(* Logix 5000 project; controller ARS14002_PLC vendor 1 type 14 code 218 rev 30.11; software revision 30.01; part 7 of 13 *)
(* tags used below, declared in another part *)
   AN_1000A : CM_AI_SCL;
   AN_1000A_SP : REAL;
   AN_1000A_SPL : REAL;
   AN_1000B : CM_AI_SCL;
   AN_1000B_SP : REAL;
   AN_1000B_SPL : REAL;
   ARGON_FROM_TK1100A : BOOL;
   ARGON_FROM_TK700 : BOOL;
   ARS_DERIME_AUTO : BOOL;
   ARS_RETURN : BOOL;
   ARS_RETURN_AUTO : BOOL;
   ARS_SOURCE_SWITCH_AUTO : BOOL;   // Switch between TK-700 and TK-1100A
   ARS_STANDBY : BOOL;
   AT2_PLANT_BACKFILL : BOOL;
   AT2_PLANT_RETURN_AUTO : BOOL;
   AT3_PLANT_BACKFILL : BOOL;
   AT3_PLANT_RETURN_AUTO : BOOL;
   Auto_CP_Select_HMI : BOOL;
   Auto_CP_Select_Inactive_ONS : BOOL;
   CP_Hi_Press_Shutoff : BOOL;
   CP_PumpUp : BOOL;
   CP_PumpUp_DN_ONS_OB : BOOL;
   CP_Run_Atomize : BOOL;
   CP_Run_ONS_OB : BOOL;
   CP_Run_ONS_SB : BOOL;
   CP_Run_Standby : BOOL;
   CP_Select_Auto : BOOL;
   CP_Select_Auto_ONS : BOOL;
   CP_Stop : BOOL;
   CP_Stop_ONS_OB : BOOL;
   CP_Stop_ONS_SB : BOOL;
   DERIME_HOLD : BOOL;
   ESTOP_TRIP : BOOL;
   ew_TEST_P800A_LOCKOUT : BOOL;
   FCV_753_SP_Idle : REAL;
   FCV_753_SP_Standby : REAL;
   FCV_754_SP_Idle : REAL;
   FCV_754_SP_Standby : REAL;
   FIRST_SCAN_BIT : BOOL;
   FT_904 : CM_AI_SCL;
   FVR_800C_Auto : BOOL;
   FVR_800C_Auto_ONS : BOOL;
   FVR_800C_AutoReq : BOOL;
   FVR_800C_ClearFault_TMR : TIMER;
   FVR_800C_DISABLE_ONS : BOOL;
   FVR_800C_EN : BOOL;
   FVR_800C_ManReq : BOOL;
   FVR_800C_ManStartReq : BOOL;
   FVR_800C_PRIMARY : BOOL;
   FVR_800C_RUNNING : BOOL;
   FVR_800C_ST : BOOL;
   FVR_800D_Auto : BOOL;
   FVR_800D_Auto_ONS : BOOL;
   FVR_800D_AutoReq : BOOL;
   FVR_800D_ClearFault_TMR : TIMER;
   FVR_800D_DISABLE_ONS : BOOL;
   FVR_800D_EN : BOOL;
   FVR_800D_ManReq : BOOL;
   FVR_800D_ManStartReq : BOOL;
   FVR_800D_PRIMARY : BOOL;
   FVR_800D_RUNNING : BOOL;
   FVR_800D_ST : BOOL;
   MODE_ATOMIZE : BOOL;
   MODE_IDLE : BOOL;
   MODE_STANDBY_IDLE : BOOL;
   MODE_STANDBY_PUMPUP : BOOL;
   P_800A_Cavit : BOOL;
   P_800A_Cooldown_Complete : BOOL;
   P_800A_Hi_Press_Shutoff : BOOL;
   P_800A_Init_OK : BOOL;
   P_800A_Pre_Vent_Done : BOOL;
   P_800A_Pre_Vent_Pending : BOOL;
   P_800A_Prestart : BOOL;
   P_800A_Ready : BOOL;
   P_800A_RUN_OCCURRED : BOOL;
   P_800A_Select_Auto_Online : BOOL;
   P_800A_Start_DLA_TMR : TIMER;
   P_800A_Start_Temp_SP : DINT;
   P_800A_Start_TMR : TIMER;
   P_800A_STOP_ONS : BOOL;
   P_800A_Stop_Vent_Delay : BOOL;
   P_800B_Cavit : BOOL;
   P_800B_Cooldown_Complete : BOOL;
   P_800B_Hi_Press_Shutoff : BOOL;
   P_800B_Init_OK : BOOL;
   P_800B_Pre_Vent_Done : BOOL;
   P_800B_Pre_Vent_Pending : BOOL;
   P_800B_Prestart : BOOL;
   P_800B_Ready : BOOL;
   P_800B_RUN_OCCURRED : BOOL;
   P_800B_Select_Auto_Online : BOOL;
   P_800B_Start_DLA_TMR : TIMER;
   P_800B_Start_Temp_SP : DINT;
   P_800B_Start_TMR : TIMER;
   P_800B_STOP_ONS : BOOL;
   P_800B_Stop_Vent_Delay : BOOL;
   P_800C : CM_DO_FVR;
   P_800C_Cavit : BOOL;
   P_800C_Cooldown_Complete : BOOL;
   P_800C_Fault : BOOL;
   P_800C_Hi_Press_Shutoff : BOOL;
   P_800C_Init_OK : BOOL;
   P_800C_Pre_Vent_Done : BOOL;
   P_800C_Pre_Vent_Pending : BOOL;
   P_800C_Prestart : BOOL;
   P_800C_Ready : BOOL;
   P_800C_RUN_OCCURRED : BOOL;
   P_800C_Select_Auto_Online : BOOL;
   P_800C_Start_DLA_TMR : TIMER;
   P_800C_Start_Temp_SP : DINT;
   P_800C_Start_TMR : TIMER;
   P_800C_STOP_ONS : BOOL;
   P_800C_Stop_Vent_Delay : BOOL;
   P_800D : CM_DO_FVR;
   P_800D_Cavit : BOOL;
   P_800D_Cooldown_Complete : BOOL;
   P_800D_Fault : BOOL;
   P_800D_Hi_Press_Shutoff : BOOL;
   P_800D_Init_OK : BOOL;
   P_800D_Pre_Vent_Done : BOOL;
   P_800D_Pre_Vent_Pending : BOOL;
   P_800D_Prestart : BOOL;
   P_800D_Ready : BOOL;
   P_800D_RUN_OCCURRED : BOOL;
   P_800D_Select_Auto_Online : BOOL;
   P_800D_Start_DLA_TMR : TIMER;
   P_800D_Start_TMR : TIMER;
   P_800D_STOP_ONS : BOOL;
   P_800D_Stop_Vent_Delay : BOOL;
   PDT_601 : CM_AI_SCL_ALT;
   PDT_701_ALT_GAL : REAL;
   PDT_751 : CM_AI_SCL_ALT;
   PIDE_753 : PID_ENHANCED;
   PIDE_754 : PID_ENHANCED;
   PIDE_755 : PID_ENHANCED;
   PIDE_800 : PID_ENHANCED;
   PILOT_PLANT_BACKFILL : BOOL;
   PILOT_PLANT_BACKFILL_COOLDOWN_DLA_SEC : REAL;
   PILOT_PLANT_BACKFILL_COOLDOWN_DLA_TMR : TIMER;   // delays the cooldown for a backfill
   PILOT_PLANT_RETURN_AUTO : BOOL;
   PT_751 : CM_AI_SCL;
   REQUEST_ARGON_FROM_TK1100A : BOOL;
   REQUEST_ARGON_FROM_TK700 : BOOL;
   SV_753F : CM_DO_GENERIC;
   SV_754F : CM_DO_GENERIC;
   SV_755F : CM_DO_GENERIC;
   TE_803_XV_721A_BURP_SP : REAL;
   TE_803A : CM_AI_SCL;
   TE_803B : CM_AI_SCL;
   TE_803C : CM_AI_SCL;
   TE_803D : CM_AI_SCL;
   TE_902 : CM_AI_SCL;
   TE_904 : CM_AI_SCL;
   TE_T_Fail_Temp : DINT;
   TEST_COOLDOWN_ALT : BOOL;
   TK_1100A_Low : BOOL;
   TK_700_AUTOFILL : BOOL;   // 1= TK-1100A WILL FILL TK-700
   TK_700_AUTOFILL_PDT_601_ALT_SPH : REAL;
   TK_700_AUTOFILL_SPH : REAL;
   TK_700_AUTOFILL_SPL : REAL;
   TK_700_AUTOSOURCE_SPH : REAL;   // Level where source will switch back to TK-700
   TK_700_AUTOSOURCE_SPL : REAL;   // Level where source will switch away from TK-700
   TK_700_FILLREQ : BOOL;
   TK_700_Full : BOOL;
   TK_700_Low : BOOL;
   VFD_800A_Auto : BOOL;
   VFD_800A_Auto_ONS : BOOL;
   VFD_800A_AutoReq : BOOL;
   VFD_800A_ClearFault_TMR : TIMER;
   VFD_800A_DISABLE_ONS : BOOL;
   VFD_800A_EN : BOOL;
   VFD_800A_ManReq : BOOL;
   VFD_800A_ManStartReq : BOOL;
   VFD_800A_ST : BOOL;
   VFD_800B_Auto : BOOL;
   VFD_800B_Auto_ONS : BOOL;
   VFD_800b_AutoReq : BOOL;
   VFD_800B_ClearFault_TMR : TIMER;
   VFD_800B_DISABLE_ONS : BOOL;
   VFD_800B_EN : BOOL;
   VFD_800B_ManReq : BOOL;
   VFD_800B_ManStartReq : BOOL;
   VFD_800B_ST : BOOL;
   XV_1123 : CM_DO_VLV;
   XV_703 : CM_DO_VLV;
   XV_721_BURP_AUTO : BOOL;
   XV_721A : CM_DO_VLV;
   XV_721B : CM_DO_VLV;
   XV_801A : CM_DO_VLV;
   XV_801B : CM_DO_VLV;
   XV_801C : CM_DO_VLV;
   XV_801D : CM_DO_VLV;
(* MainProgram, continued *)

ROUTINE _304_Subcooler   (* ladder *)
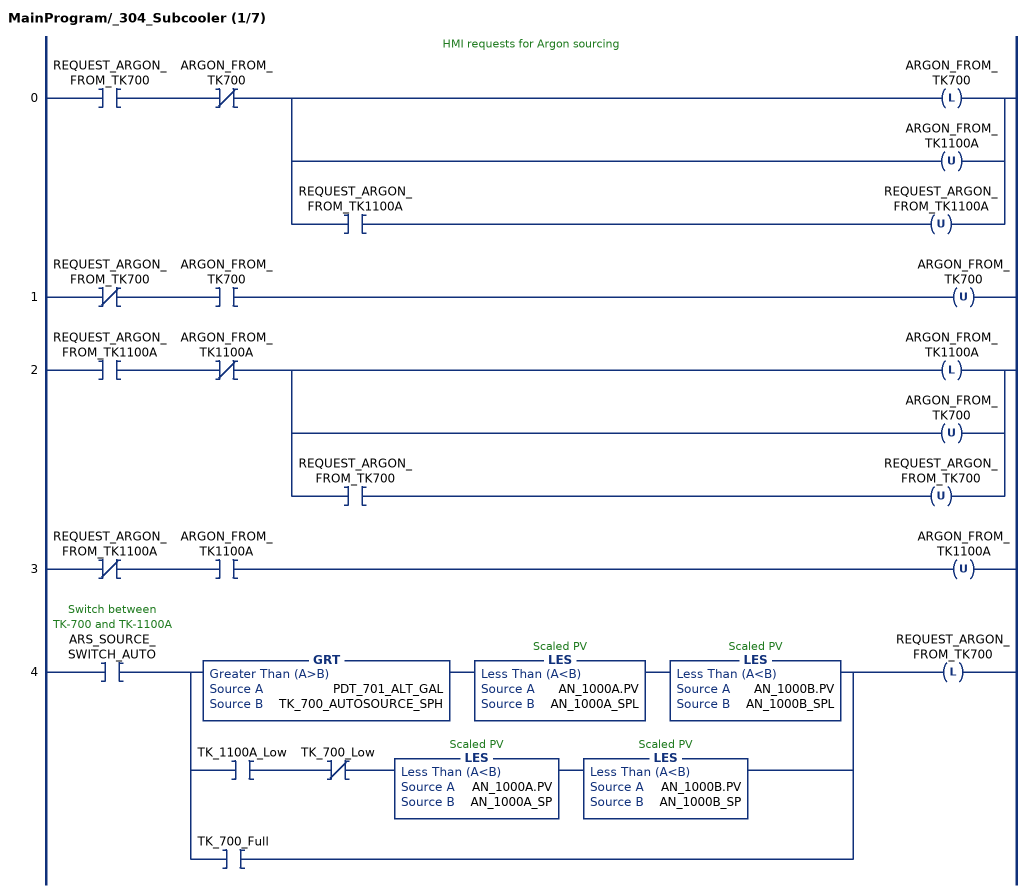
   // HMI requests for Argon sourcing
   0: XIC(REQUEST_ARGON_FROM_TK700)XIO(ARGON_FROM_TK700)[OTL(ARGON_FROM_TK700) ,OTU(ARGON_FROM_TK1100A) ,XIC(REQUEST_ARGON_FROM_TK1100A) OTU(REQUEST_ARGON_FROM_TK1100A) ];
   1: XIO(REQUEST_ARGON_FROM_TK700)XIC(ARGON_FROM_TK700)OTU(ARGON_FROM_TK700);
   2: XIC(REQUEST_ARGON_FROM_TK1100A)XIO(ARGON_FROM_TK1100A)[OTL(ARGON_FROM_TK1100A) ,OTU(ARGON_FROM_TK700) ,XIC(REQUEST_ARGON_FROM_TK700) OTU(REQUEST_ARGON_FROM_TK700) ];
   3: XIO(REQUEST_ARGON_FROM_TK1100A)XIC(ARGON_FROM_TK1100A)OTU(ARGON_FROM_TK1100A);
   4: XIC(ARS_SOURCE_SWITCH_AUTO)[GRT(PDT_701_ALT_GAL,TK_700_AUTOSOURCE_SPH) LES(AN_1000A.PV,AN_1000A_SPL) LES(AN_1000B.PV,AN_1000B_SPL) ,XIC(TK_1100A_Low) XIO(TK_700_Low) LES(AN_1000A.PV,AN_1000A_SP) LES(AN_1000B.PV,AN_1000B_SP) ,XIC(TK_700_Full) ]OTL(REQUEST_ARGON_FROM_TK700);
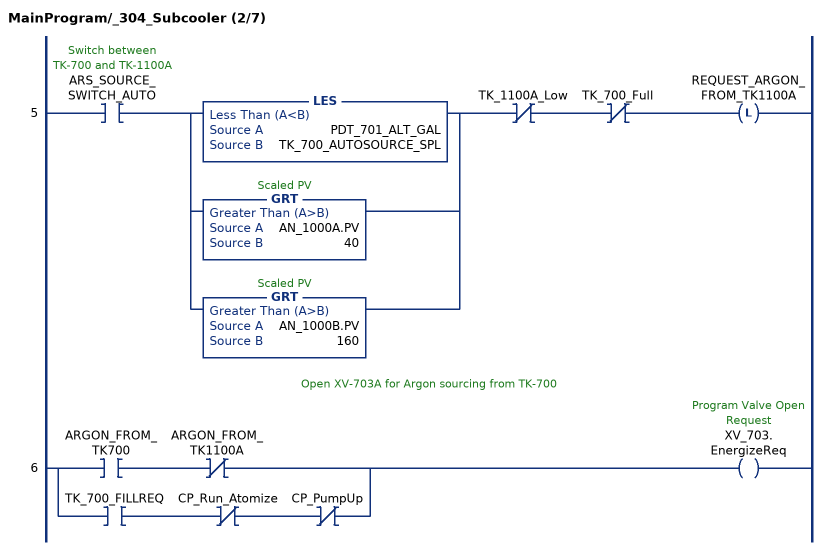
   5: XIC(ARS_SOURCE_SWITCH_AUTO)[LES(PDT_701_ALT_GAL,TK_700_AUTOSOURCE_SPL) ,GRT(AN_1000A.PV,40) ,GRT(AN_1000B.PV,160) ]XIO(TK_1100A_Low)XIO(TK_700_Full)OTL(REQUEST_ARGON_FROM_TK1100A);
   // Open XV-703A for Argon sourcing from TK-700
   6: [XIC(ARGON_FROM_TK700) XIO(ARGON_FROM_TK1100A) ,XIC(TK_700_FILLREQ) XIO(CP_Run_Atomize) XIO(CP_PumpUp) ]OTE(XV_703.EnergizeReq);
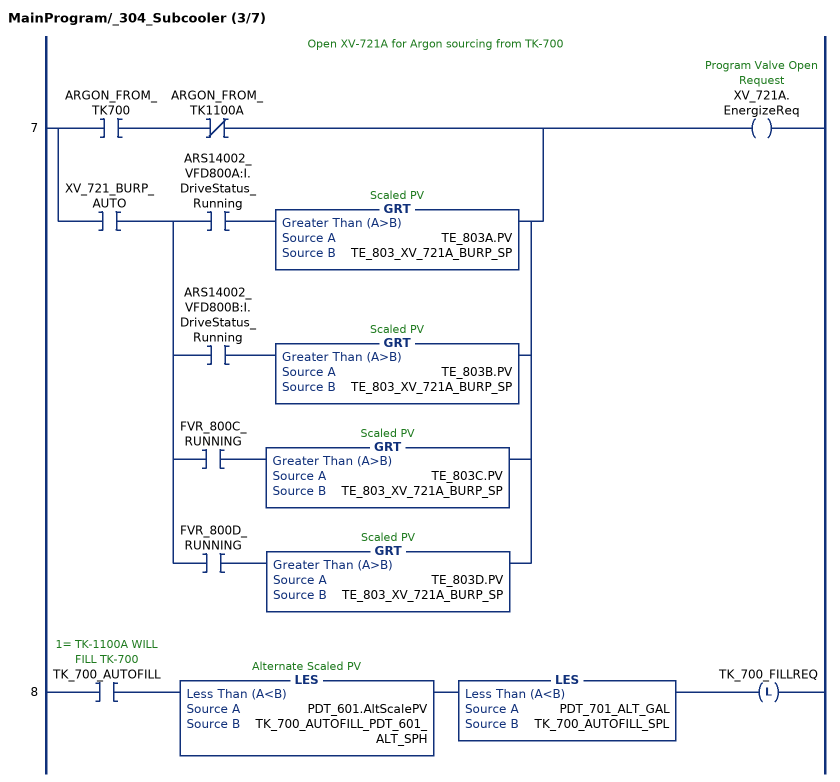
   // Open XV-721A for Argon sourcing from TK-700
   7: [XIC(ARGON_FROM_TK700) XIO(ARGON_FROM_TK1100A) ,XIC(XV_721_BURP_AUTO) [XIC(ARS14002_VFD800A:I.DriveStatus_Running) GRT(TE_803A.PV,TE_803_XV_721A_BURP_SP) ,XIC(ARS14002_VFD800B:I.DriveStatus_Running) GRT(TE_803B.PV,TE_803_XV_721A_BURP_SP) ,XIC(FVR_800C_RUNNING) GRT(TE_803C.PV,TE_803_XV_721A_BURP_SP) ,XIC(FVR_800D_RUNNING) GRT(TE_803D.PV,TE_803_XV_721A_BURP_SP) ] ]OTE(XV_721A.EnergizeReq);
   8: XIC(TK_700_AUTOFILL)LES(PDT_601.AltScalePV,TK_700_AUTOFILL_PDT_601_ALT_SPH)LES(PDT_701_ALT_GAL,TK_700_AUTOFILL_SPL)OTL(TK_700_FILLREQ);
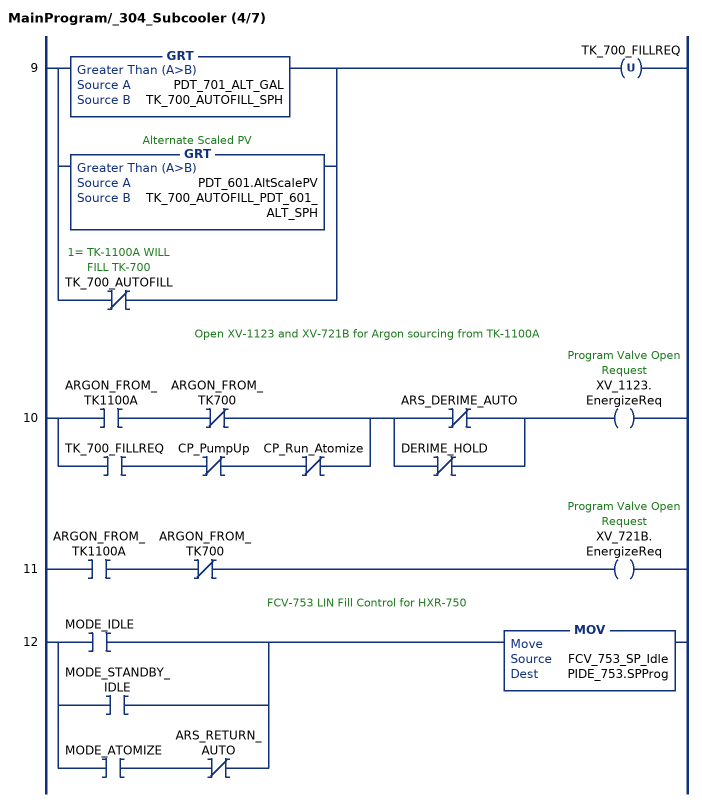
   9: [GRT(PDT_701_ALT_GAL,TK_700_AUTOFILL_SPH) ,GRT(PDT_601.AltScalePV,TK_700_AUTOFILL_PDT_601_ALT_SPH) ,XIO(TK_700_AUTOFILL) ]OTU(TK_700_FILLREQ);
   // Open XV-1123 and XV-721B for Argon sourcing from TK-1100A
   10: [XIC(ARGON_FROM_TK1100A) XIO(ARGON_FROM_TK700) ,XIC(TK_700_FILLREQ) XIO(CP_PumpUp) XIO(CP_Run_Atomize) ][XIO(ARS_DERIME_AUTO) ,XIO(DERIME_HOLD) ]OTE(XV_1123.EnergizeReq);
   11: XIC(ARGON_FROM_TK1100A)XIO(ARGON_FROM_TK700)OTE(XV_721B.EnergizeReq);
   // FCV-753 LIN Fill Control for HXR-750
   12: [XIC(MODE_IDLE) ,XIC(MODE_STANDBY_IDLE) ,XIC(MODE_ATOMIZE) XIO(ARS_RETURN_AUTO) ]MOV(FCV_753_SP_Idle,PIDE_753.SPProg);
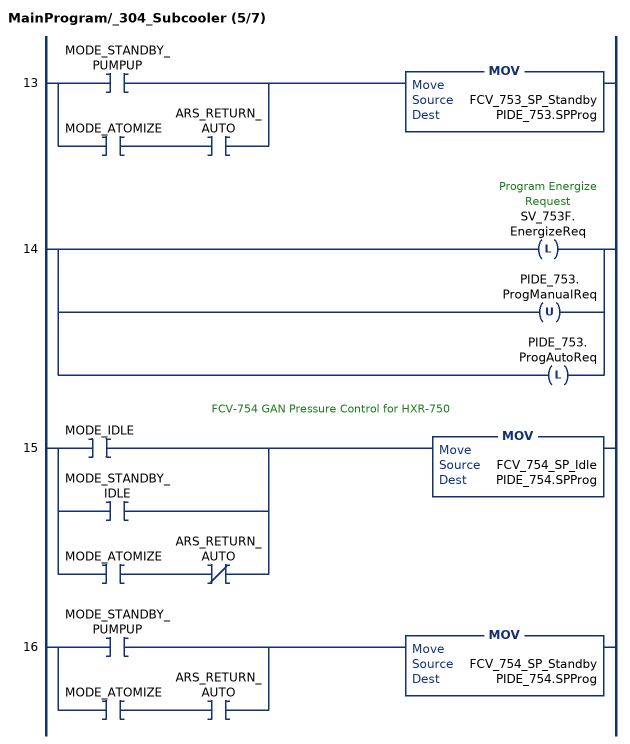
   13: [XIC(MODE_STANDBY_PUMPUP) ,XIC(MODE_ATOMIZE) XIC(ARS_RETURN_AUTO) ]MOV(FCV_753_SP_Standby,PIDE_753.SPProg);
   14: [OTL(SV_753F.EnergizeReq) ,OTU(PIDE_753.ProgManualReq) ,OTL(PIDE_753.ProgAutoReq) ];
   // FCV-754 GAN Pressure Control for HXR-750
   15: [XIC(MODE_IDLE) ,XIC(MODE_STANDBY_IDLE) ,XIC(MODE_ATOMIZE) XIO(ARS_RETURN_AUTO) ]MOV(FCV_754_SP_Idle,PIDE_754.SPProg);
   16: [XIC(MODE_STANDBY_PUMPUP) ,XIC(MODE_ATOMIZE) XIC(ARS_RETURN_AUTO) ]MOV(FCV_754_SP_Standby,PIDE_754.SPProg);
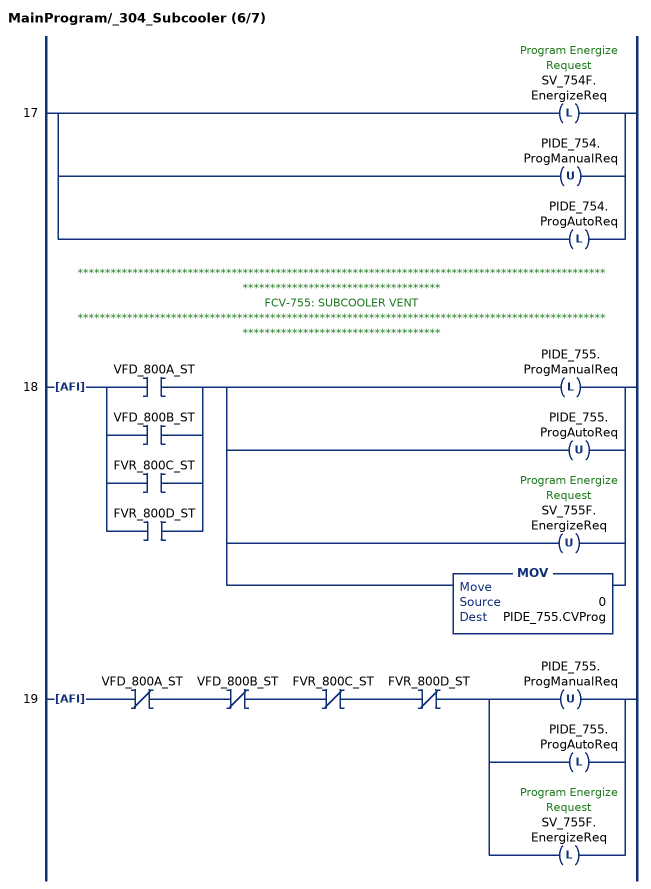
   17: [OTL(SV_754F.EnergizeReq) ,OTU(PIDE_754.ProgManualReq) ,OTL(PIDE_754.ProgAutoReq) ];
   // ************************************************************************************************************************************
   // FCV-755: SUBCOOLER VENT
   // ************************************************************************************************************************************
   18: AFI()[XIC(VFD_800A_ST) ,XIC(VFD_800B_ST) ,XIC(FVR_800C_ST) ,XIC(FVR_800D_ST) ][OTL(PIDE_755.ProgManualReq) ,OTU(PIDE_755.ProgAutoReq) ,OTU(SV_755F.EnergizeReq) ,MOV(0,PIDE_755.CVProg) ];
   19: AFI()XIO(VFD_800A_ST)XIO(VFD_800B_ST)XIO(FVR_800C_ST)XIO(FVR_800D_ST)[OTU(PIDE_755.ProgManualReq) ,OTL(PIDE_755.ProgAutoReq) ,OTL(SV_755F.EnergizeReq) ];
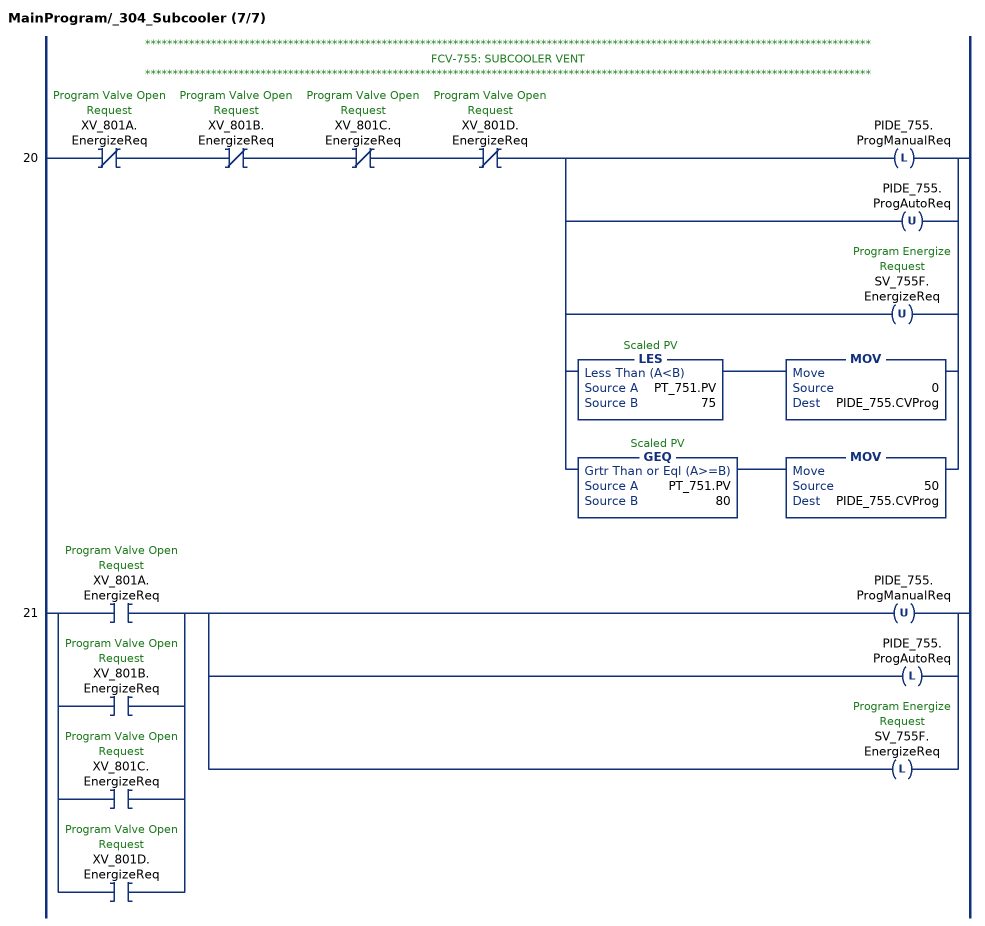
   // ************************************************************************************************************************************
   // FCV-755: SUBCOOLER VENT
   // ************************************************************************************************************************************
   20: XIO(XV_801A.EnergizeReq)XIO(XV_801B.EnergizeReq)XIO(XV_801C.EnergizeReq)XIO(XV_801D.EnergizeReq)[OTL(PIDE_755.ProgManualReq) ,OTU(PIDE_755.ProgAutoReq) ,OTU(SV_755F.EnergizeReq) ,LES(PT_751.PV,75) MOV(0,PIDE_755.CVProg) ,GEQ(PT_751.PV,80) MOV(50,PIDE_755.CVProg) ];
   21: [XIC(XV_801A.EnergizeReq) ,XIC(XV_801B.EnergizeReq) ,XIC(XV_801C.EnergizeReq) ,XIC(XV_801D.EnergizeReq) ][OTU(PIDE_755.ProgManualReq) ,OTL(PIDE_755.ProgAutoReq) ,OTL(SV_755F.EnergizeReq) ];
END_ROUTINE

ROUTINE _305_Pump_800   (* ladder *)
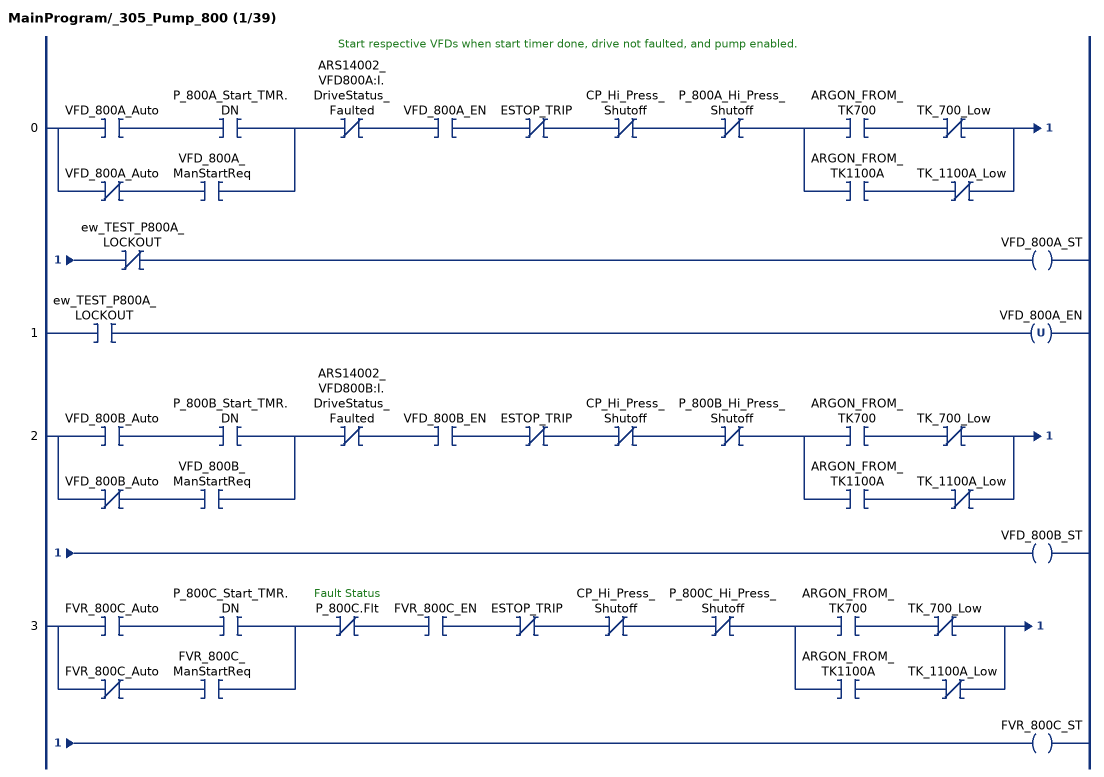
   // Start respective VFDs when start timer done, drive not faulted, and pump enabled.
   0: [XIC(VFD_800A_Auto) XIC(P_800A_Start_TMR.DN) ,XIO(VFD_800A_Auto) XIC(VFD_800A_ManStartReq) ]XIO(ARS14002_VFD800A:I.DriveStatus_Faulted)XIC(VFD_800A_EN)XIO(ESTOP_TRIP)XIO(CP_Hi_Press_Shutoff)XIO(P_800A_Hi_Press_Shutoff)[XIC(ARGON_FROM_TK700) XIO(TK_700_Low) ,XIC(ARGON_FROM_TK1100A) XIO(TK_1100A_Low) ]XIO(ew_TEST_P800A_LOCKOUT)OTE(VFD_800A_ST);
   1: XIC(ew_TEST_P800A_LOCKOUT)OTU(VFD_800A_EN);
   2: [XIC(VFD_800B_Auto) XIC(P_800B_Start_TMR.DN) ,XIO(VFD_800B_Auto) XIC(VFD_800B_ManStartReq) ]XIO(ARS14002_VFD800B:I.DriveStatus_Faulted)XIC(VFD_800B_EN)XIO(ESTOP_TRIP)XIO(CP_Hi_Press_Shutoff)XIO(P_800B_Hi_Press_Shutoff)[XIC(ARGON_FROM_TK700) XIO(TK_700_Low) ,XIC(ARGON_FROM_TK1100A) XIO(TK_1100A_Low) ]OTE(VFD_800B_ST);
   3: [XIC(FVR_800C_Auto) XIC(P_800C_Start_TMR.DN) ,XIO(FVR_800C_Auto) XIC(FVR_800C_ManStartReq) ]XIO(P_800C.Flt)XIC(FVR_800C_EN)XIO(ESTOP_TRIP)XIO(CP_Hi_Press_Shutoff)XIO(P_800C_Hi_Press_Shutoff)[XIC(ARGON_FROM_TK700) XIO(TK_700_Low) ,XIC(ARGON_FROM_TK1100A) XIO(TK_1100A_Low) ]OTE(FVR_800C_ST);
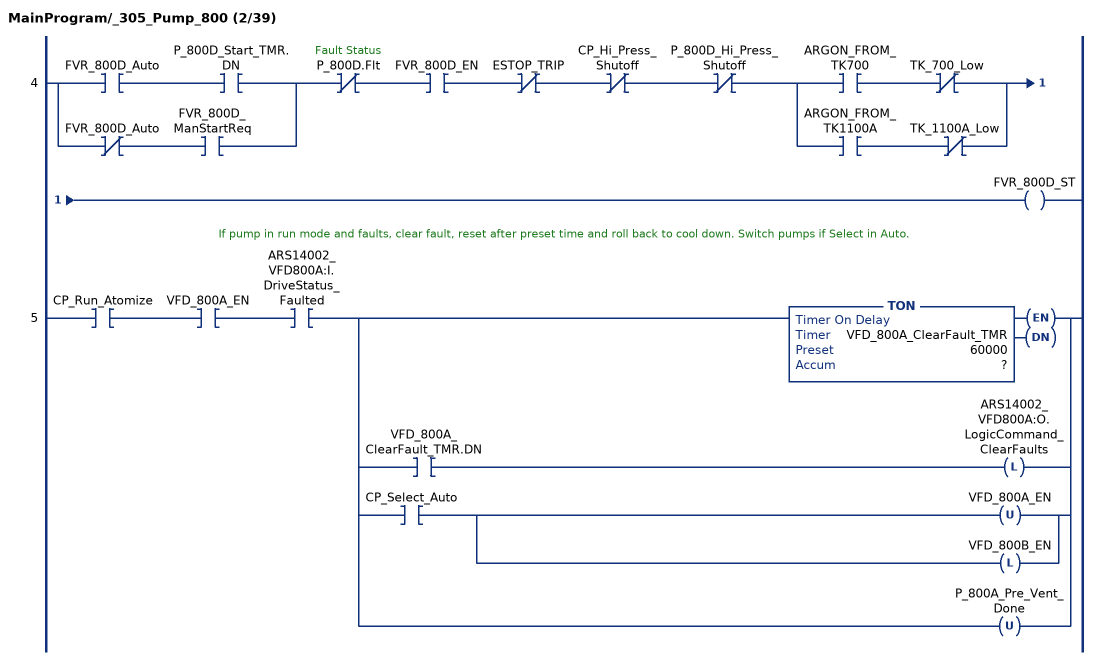
   4: [XIC(FVR_800D_Auto) XIC(P_800D_Start_TMR.DN) ,XIO(FVR_800D_Auto) XIC(FVR_800D_ManStartReq) ]XIO(P_800D.Flt)XIC(FVR_800D_EN)XIO(ESTOP_TRIP)XIO(CP_Hi_Press_Shutoff)XIO(P_800D_Hi_Press_Shutoff)[XIC(ARGON_FROM_TK700) XIO(TK_700_Low) ,XIC(ARGON_FROM_TK1100A) XIO(TK_1100A_Low) ]OTE(FVR_800D_ST);
   // If pump in run mode and faults, clear fault, reset after preset time and roll back to cool down. Switch pumps if Select in Auto.
   5: XIC(CP_Run_Atomize)XIC(VFD_800A_EN)XIC(ARS14002_VFD800A:I.DriveStatus_Faulted)[[TON(VFD_800A_ClearFault_TMR,?,?) ,XIC(VFD_800A_ClearFault_TMR.DN) OTL(ARS14002_VFD800A:O.LogicCommand_ClearFaults) ,XIC(CP_Select_Auto) [OTU(VFD_800A_EN) ,OTL(VFD_800B_EN) ] ] ,OTU(P_800A_Pre_Vent_Done) ];
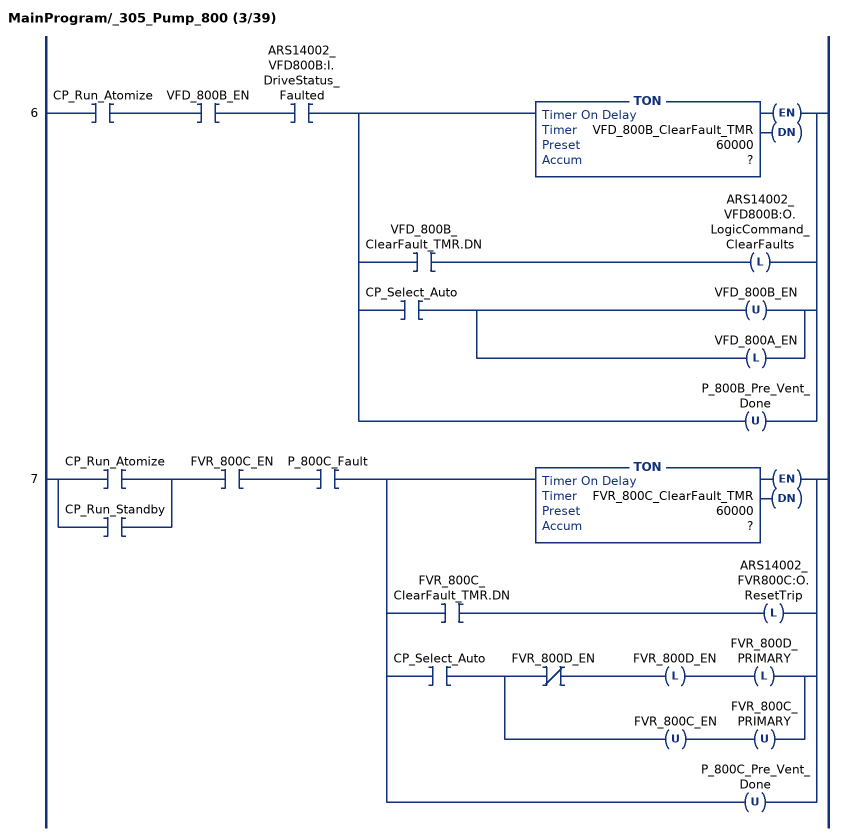
   6: XIC(CP_Run_Atomize)XIC(VFD_800B_EN)XIC(ARS14002_VFD800B:I.DriveStatus_Faulted)[[TON(VFD_800B_ClearFault_TMR,?,?) ,XIC(VFD_800B_ClearFault_TMR.DN) OTL(ARS14002_VFD800B:O.LogicCommand_ClearFaults) ,XIC(CP_Select_Auto) [OTU(VFD_800B_EN) ,OTL(VFD_800A_EN) ] ] ,OTU(P_800B_Pre_Vent_Done) ];
   7: [XIC(CP_Run_Atomize) ,XIC(CP_Run_Standby) ]XIC(FVR_800C_EN)XIC(P_800C_Fault)[[TON(FVR_800C_ClearFault_TMR,?,?) ,XIC(FVR_800C_ClearFault_TMR.DN) OTL(ARS14002_FVR800C:O.ResetTrip) ,XIC(CP_Select_Auto) [XIO(FVR_800D_EN) OTL(FVR_800D_EN) OTL(FVR_800D_PRIMARY) ,OTU(FVR_800C_EN) OTU(FVR_800C_PRIMARY) ] ] ,OTU(P_800C_Pre_Vent_Done) ];
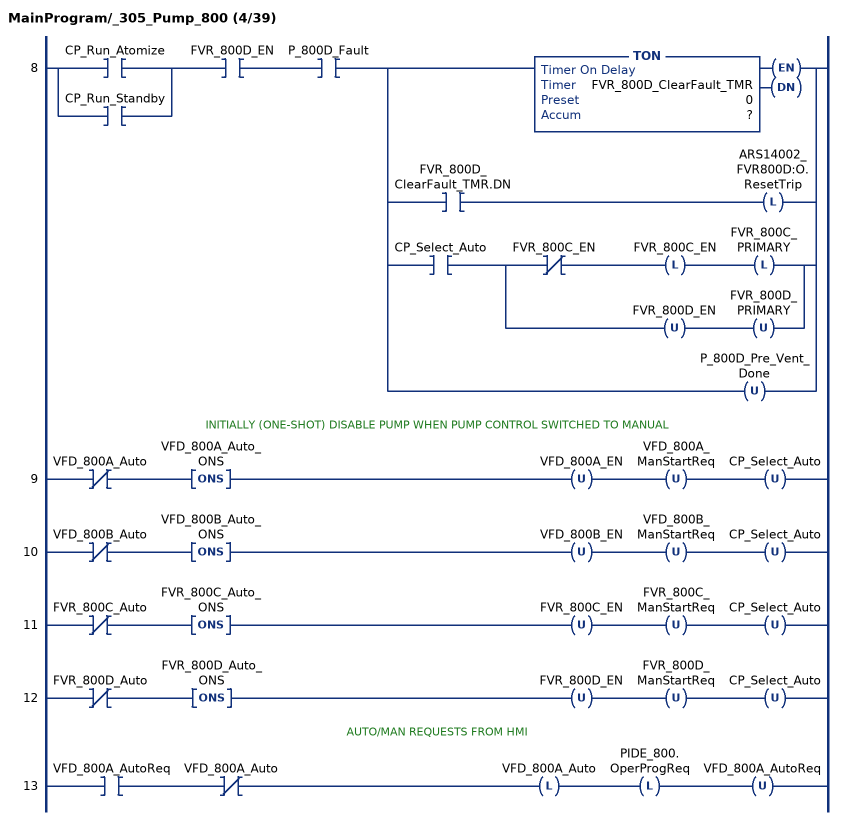
   8: [XIC(CP_Run_Atomize) ,XIC(CP_Run_Standby) ]XIC(FVR_800D_EN)XIC(P_800D_Fault)[[TON(FVR_800D_ClearFault_TMR,?,?) ,XIC(FVR_800D_ClearFault_TMR.DN) OTL(ARS14002_FVR800D:O.ResetTrip) ,XIC(CP_Select_Auto) [XIO(FVR_800C_EN) OTL(FVR_800C_EN) OTL(FVR_800C_PRIMARY) ,OTU(FVR_800D_EN) OTU(FVR_800D_PRIMARY) ] ] ,OTU(P_800D_Pre_Vent_Done) ];
   // INITIALLY (ONE-SHOT) DISABLE PUMP WHEN PUMP CONTROL SWITCHED TO MANUAL
   9: XIO(VFD_800A_Auto)ONS(VFD_800A_Auto_ONS)OTU(VFD_800A_EN)OTU(VFD_800A_ManStartReq)OTU(CP_Select_Auto);
   10: XIO(VFD_800B_Auto)ONS(VFD_800B_Auto_ONS)OTU(VFD_800B_EN)OTU(VFD_800B_ManStartReq)OTU(CP_Select_Auto);
   11: XIO(FVR_800C_Auto)ONS(FVR_800C_Auto_ONS)OTU(FVR_800C_EN)OTU(FVR_800C_ManStartReq)OTU(CP_Select_Auto);
   12: XIO(FVR_800D_Auto)ONS(FVR_800D_Auto_ONS)OTU(FVR_800D_EN)OTU(FVR_800D_ManStartReq)OTU(CP_Select_Auto);
   // AUTO/MAN REQUESTS FROM HMI
   13: XIC(VFD_800A_AutoReq)XIO(VFD_800A_Auto)OTL(VFD_800A_Auto)OTL(PIDE_800.OperProgReq)OTU(VFD_800A_AutoReq);
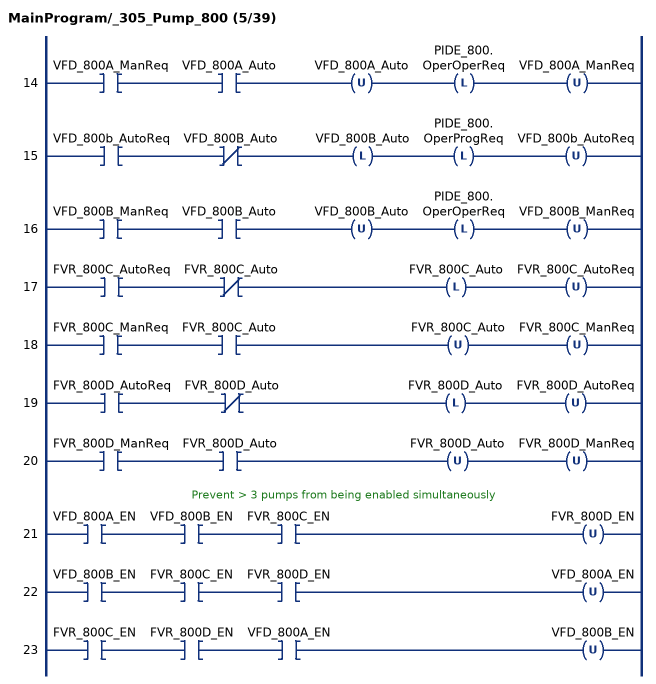
   14: XIC(VFD_800A_ManReq)XIC(VFD_800A_Auto)OTU(VFD_800A_Auto)OTL(PIDE_800.OperOperReq)OTU(VFD_800A_ManReq);
   15: XIC(VFD_800b_AutoReq)XIO(VFD_800B_Auto)OTL(VFD_800B_Auto)OTL(PIDE_800.OperProgReq)OTU(VFD_800b_AutoReq);
   16: XIC(VFD_800B_ManReq)XIC(VFD_800B_Auto)OTU(VFD_800B_Auto)OTL(PIDE_800.OperOperReq)OTU(VFD_800B_ManReq);
   17: XIC(FVR_800C_AutoReq)XIO(FVR_800C_Auto)OTL(FVR_800C_Auto)OTU(FVR_800C_AutoReq);
   18: XIC(FVR_800C_ManReq)XIC(FVR_800C_Auto)OTU(FVR_800C_Auto)OTU(FVR_800C_ManReq);
   19: XIC(FVR_800D_AutoReq)XIO(FVR_800D_Auto)OTL(FVR_800D_Auto)OTU(FVR_800D_AutoReq);
   20: XIC(FVR_800D_ManReq)XIC(FVR_800D_Auto)OTU(FVR_800D_Auto)OTU(FVR_800D_ManReq);
   // Prevent > 3 pumps from being enabled simultaneously
   21: XIC(VFD_800A_EN)XIC(VFD_800B_EN)XIC(FVR_800C_EN)OTU(FVR_800D_EN);
   22: XIC(VFD_800B_EN)XIC(FVR_800C_EN)XIC(FVR_800D_EN)OTU(VFD_800A_EN);
   23: XIC(FVR_800C_EN)XIC(FVR_800D_EN)XIC(VFD_800A_EN)OTU(VFD_800B_EN);
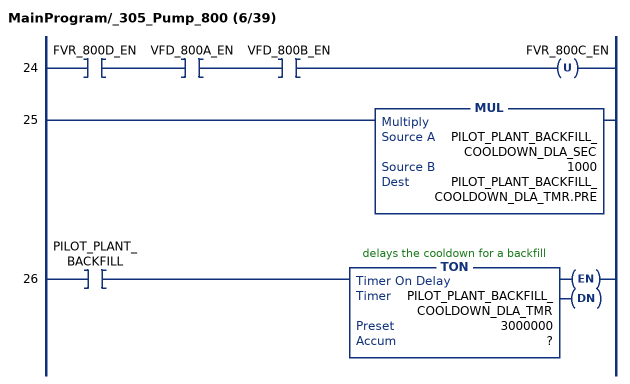
   24: XIC(FVR_800D_EN)XIC(VFD_800A_EN)XIC(VFD_800B_EN)OTU(FVR_800C_EN);
   25: MUL(PILOT_PLANT_BACKFILL_COOLDOWN_DLA_SEC,1000,PILOT_PLANT_BACKFILL_COOLDOWN_DLA_TMR.PRE);
   26: XIC(PILOT_PLANT_BACKFILL)TON(PILOT_PLANT_BACKFILL_COOLDOWN_DLA_TMR,?,?);
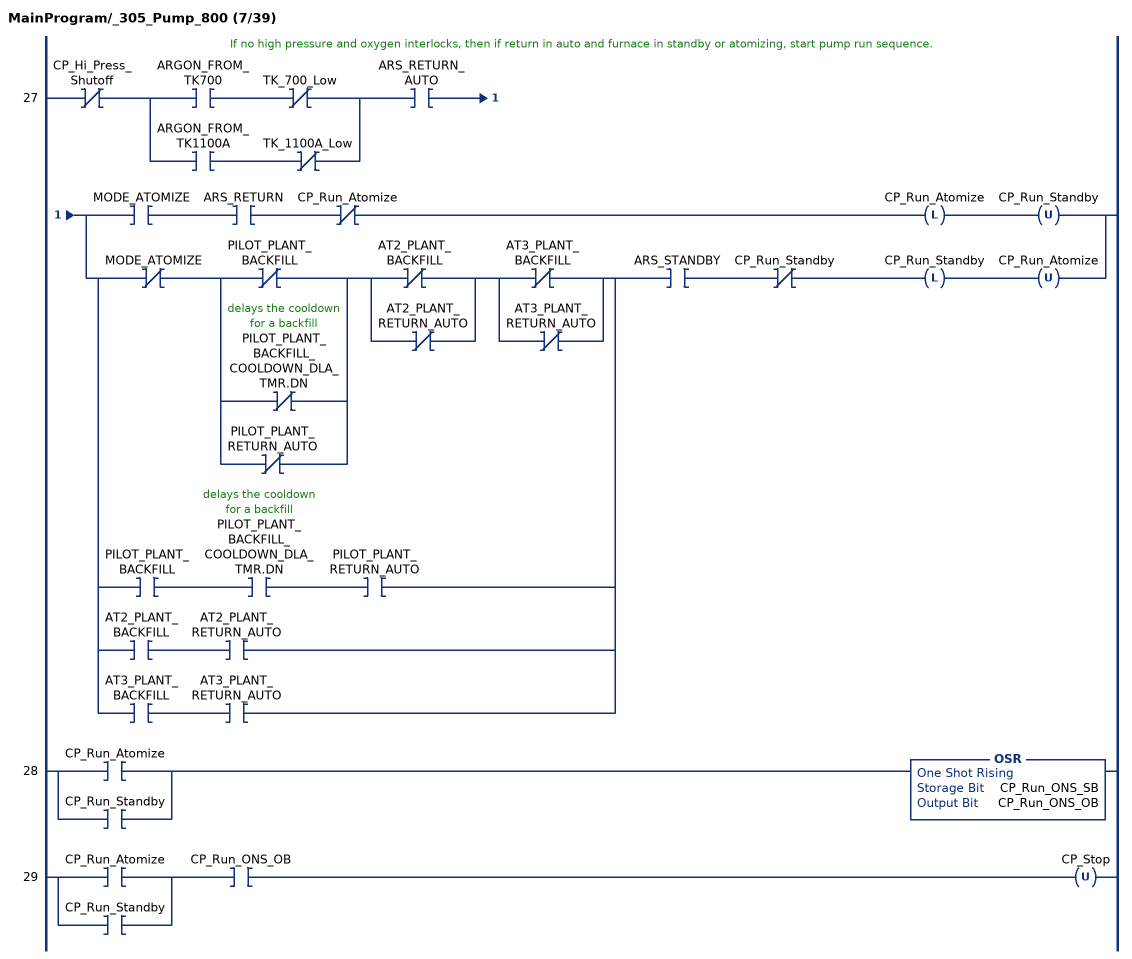
   // If no high pressure and oxygen interlocks, then if return in auto and furnace in standby or atomizing, start pump run sequence.
   27: XIO(CP_Hi_Press_Shutoff)[XIC(ARGON_FROM_TK700) XIO(TK_700_Low) ,XIC(ARGON_FROM_TK1100A) XIO(TK_1100A_Low) ]XIC(ARS_RETURN_AUTO)[XIC(MODE_ATOMIZE) XIC(ARS_RETURN) XIO(CP_Run_Atomize) OTL(CP_Run_Atomize) OTU(CP_Run_Standby) ,[XIO(MODE_ATOMIZE) [XIO(PILOT_PLANT_BACKFILL) ,XIO(PILOT_PLANT_BACKFILL_COOLDOWN_DLA_TMR.DN) ,XIO(PILOT_PLANT_RETURN_AUTO) ] [XIO(AT2_PLANT_BACKFILL) ,XIO(AT2_PLANT_RETURN_AUTO) ] [XIO(AT3_PLANT_BACKFILL) ,XIO(AT3_PLANT_RETURN_AUTO) ] ,XIC(PILOT_PLANT_BACKFILL) XIC(PILOT_PLANT_BACKFILL_COOLDOWN_DLA_TMR.DN) XIC(PILOT_PLANT_RETURN_AUTO) ,XIC(AT2_PLANT_BACKFILL) XIC(AT2_PLANT_RETURN_AUTO) ,XIC(AT3_PLANT_BACKFILL) XIC(AT3_PLANT_RETURN_AUTO) ] XIC(ARS_STANDBY) XIO(CP_Run_Standby) OTL(CP_Run_Standby) OTU(CP_Run_Atomize) ];
   28: [XIC(CP_Run_Atomize) ,XIC(CP_Run_Standby) ]OSR(CP_Run_ONS_SB,CP_Run_ONS_OB);
   29: [XIC(CP_Run_Atomize) ,XIC(CP_Run_Standby) ]XIC(CP_Run_ONS_OB)OTU(CP_Stop);
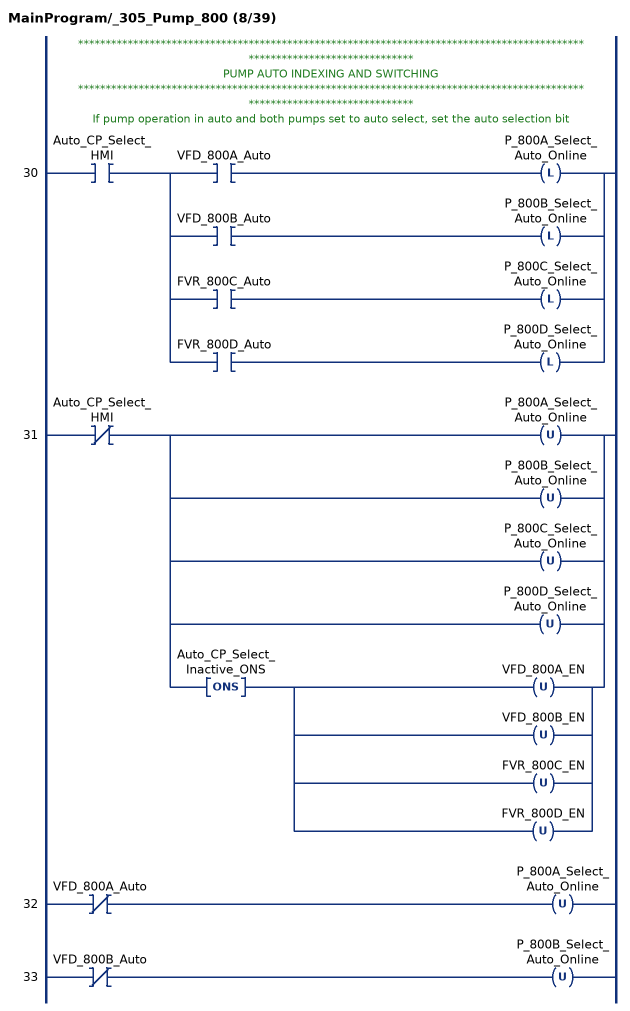
   // **************************************************************************************************************************
   // PUMP AUTO INDEXING AND SWITCHING
   // **************************************************************************************************************************
   // If pump operation in auto and both pumps set to auto select, set the auto selection bit
   30: XIC(Auto_CP_Select_HMI)[XIC(VFD_800A_Auto) OTL(P_800A_Select_Auto_Online) ,XIC(VFD_800B_Auto) OTL(P_800B_Select_Auto_Online) ,XIC(FVR_800C_Auto) OTL(P_800C_Select_Auto_Online) ,XIC(FVR_800D_Auto) OTL(P_800D_Select_Auto_Online) ];
   31: XIO(Auto_CP_Select_HMI)[[OTU(P_800A_Select_Auto_Online) ,OTU(P_800B_Select_Auto_Online) ,OTU(P_800C_Select_Auto_Online) ,OTU(P_800D_Select_Auto_Online) ] ,ONS(Auto_CP_Select_Inactive_ONS) [OTU(VFD_800A_EN) ,OTU(VFD_800B_EN) ,OTU(FVR_800C_EN) ,OTU(FVR_800D_EN) ] ];
   32: XIO(VFD_800A_Auto)OTU(P_800A_Select_Auto_Online);
   33: XIO(VFD_800B_Auto)OTU(P_800B_Select_Auto_Online);
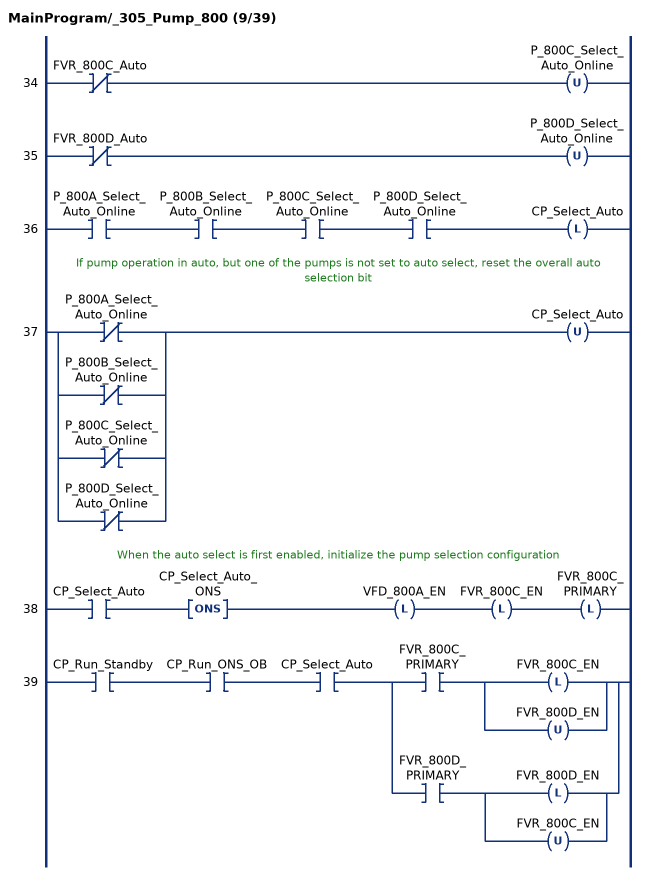
   34: XIO(FVR_800C_Auto)OTU(P_800C_Select_Auto_Online);
   35: XIO(FVR_800D_Auto)OTU(P_800D_Select_Auto_Online);
   36: XIC(P_800A_Select_Auto_Online)XIC(P_800B_Select_Auto_Online)XIC(P_800C_Select_Auto_Online)XIC(P_800D_Select_Auto_Online)OTL(CP_Select_Auto);
   // If pump operation in auto, but one of the pumps is not set to auto select, reset the overall auto selection bit
   37: [XIO(P_800A_Select_Auto_Online) ,XIO(P_800B_Select_Auto_Online) ,XIO(P_800C_Select_Auto_Online) ,XIO(P_800D_Select_Auto_Online) ]OTU(CP_Select_Auto);
   // When the auto select is first enabled, initialize the pump selection configuration
   38: XIC(CP_Select_Auto)ONS(CP_Select_Auto_ONS)OTL(VFD_800A_EN)OTL(FVR_800C_EN)OTL(FVR_800C_PRIMARY);
   39: XIC(CP_Run_Standby)XIC(CP_Run_ONS_OB)XIC(CP_Select_Auto)[XIC(FVR_800C_PRIMARY) [OTL(FVR_800C_EN) ,OTU(FVR_800D_EN) ] ,XIC(FVR_800D_PRIMARY) [OTL(FVR_800D_EN) ,OTU(FVR_800C_EN) ] ];
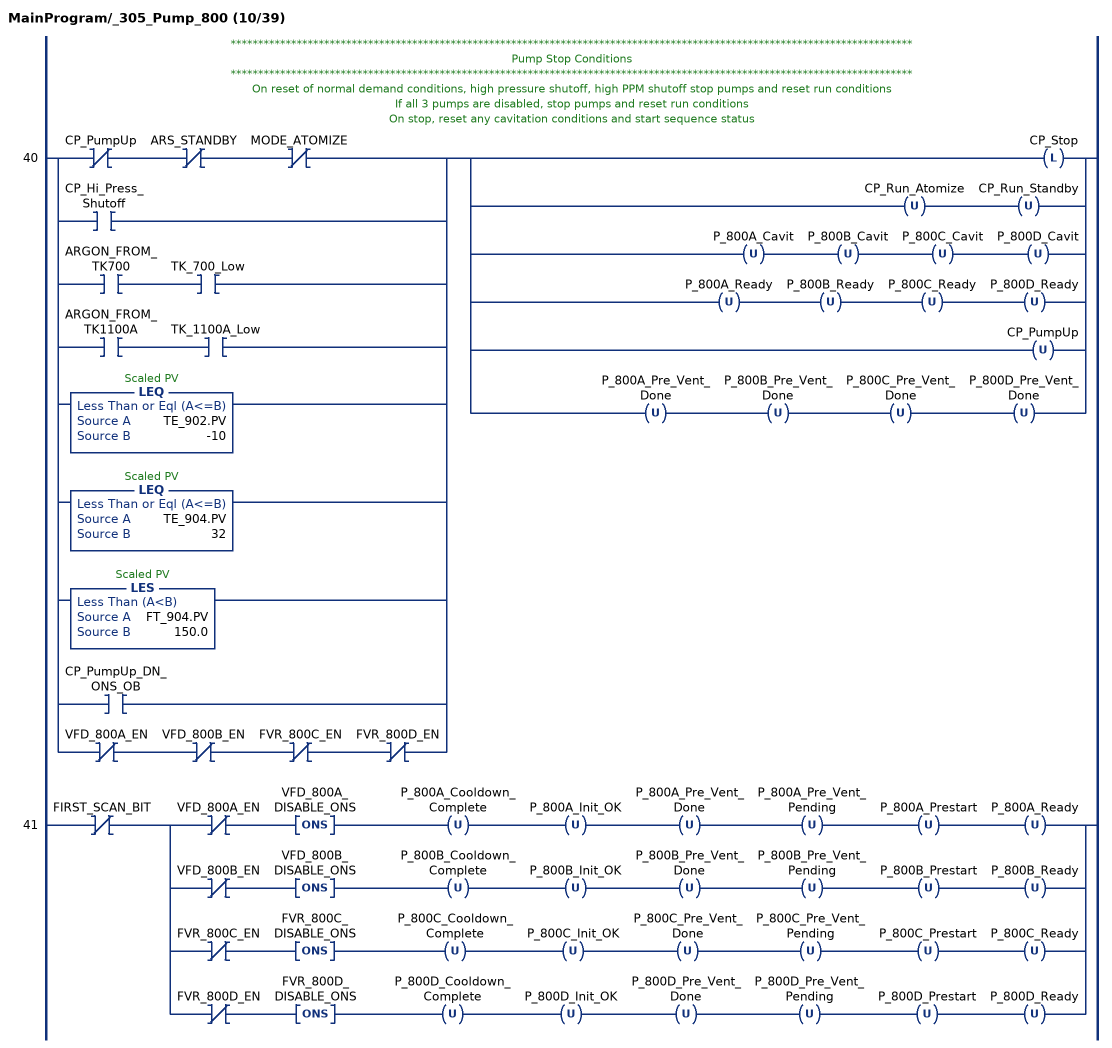
   // ****************************************************************************************************************************
   // Pump Stop Conditions
   // ****************************************************************************************************************************
   // On reset of normal demand conditions, high pressure shutoff, high PPM shutoff stop pumps and reset run conditions
   // If all 3 pumps are disabled, stop pumps and reset run conditions
   // On stop, reset any cavitation conditions and start sequence status
   40: [XIO(CP_PumpUp) XIO(ARS_STANDBY) XIO(MODE_ATOMIZE) ,XIC(CP_Hi_Press_Shutoff) ,XIC(ARGON_FROM_TK700) XIC(TK_700_Low) ,XIC(ARGON_FROM_TK1100A) XIC(TK_1100A_Low) ,LEQ(TE_902.PV,-10) ,LEQ(TE_904.PV,32) ,LES(FT_904.PV,150.0) ,XIC(CP_PumpUp_DN_ONS_OB) ,XIO(VFD_800A_EN) XIO(VFD_800B_EN) XIO(FVR_800C_EN) XIO(FVR_800D_EN) ][OTL(CP_Stop) ,OTU(CP_Run_Atomize) OTU(CP_Run_Standby) ,OTU(P_800A_Cavit) OTU(P_800B_Cavit) OTU(P_800C_Cavit) OTU(P_800D_Cavit) ,OTU(P_800A_Ready) OTU(P_800B_Ready) OTU(P_800C_Ready) OTU(P_800D_Ready) ,OTU(CP_PumpUp) ,OTU(P_800A_Pre_Vent_Done) OTU(P_800B_Pre_Vent_Done) OTU(P_800C_Pre_Vent_Done) OTU(P_800D_Pre_Vent_Done) ];
   41: XIO(FIRST_SCAN_BIT)[XIO(VFD_800A_EN) ONS(VFD_800A_DISABLE_ONS) OTU(P_800A_Cooldown_Complete) OTU(P_800A_Init_OK) OTU(P_800A_Pre_Vent_Done) OTU(P_800A_Pre_Vent_Pending) OTU(P_800A_Prestart) OTU(P_800A_Ready) ,XIO(VFD_800B_EN) ONS(VFD_800B_DISABLE_ONS) OTU(P_800B_Cooldown_Complete) OTU(P_800B_Init_OK) OTU(P_800B_Pre_Vent_Done) OTU(P_800B_Pre_Vent_Pending) OTU(P_800B_Prestart) OTU(P_800B_Ready) ,XIO(FVR_800C_EN) ONS(FVR_800C_DISABLE_ONS) OTU(P_800C_Cooldown_Complete) OTU(P_800C_Init_OK) OTU(P_800C_Pre_Vent_Done) OTU(P_800C_Pre_Vent_Pending) OTU(P_800C_Prestart) OTU(P_800C_Ready) ,XIO(FVR_800D_EN) ONS(FVR_800D_DISABLE_ONS) OTU(P_800D_Cooldown_Complete) OTU(P_800D_Init_OK) OTU(P_800D_Pre_Vent_Done) OTU(P_800D_Pre_Vent_Pending) OTU(P_800D_Prestart) OTU(P_800D_Ready) ];
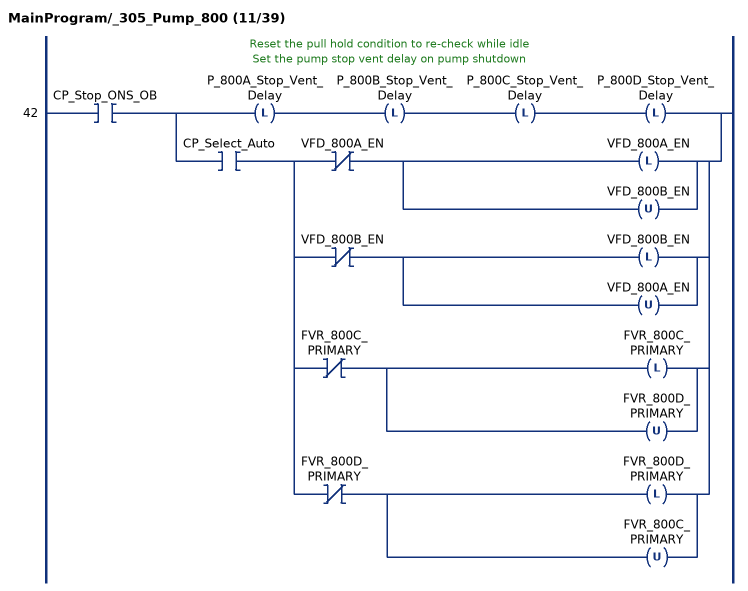
   // Reset the pull hold condition to re-check while idle
   // Set the pump stop vent delay on pump shutdown
   42: XIC(CP_Stop_ONS_OB)[OTL(P_800A_Stop_Vent_Delay) OTL(P_800B_Stop_Vent_Delay) OTL(P_800C_Stop_Vent_Delay) OTL(P_800D_Stop_Vent_Delay) ,XIC(CP_Select_Auto) [XIO(VFD_800A_EN) [OTL(VFD_800A_EN) ,OTU(VFD_800B_EN) ] ,XIO(VFD_800B_EN) [OTL(VFD_800B_EN) ,OTU(VFD_800A_EN) ] ,XIO(FVR_800C_PRIMARY) [OTL(FVR_800C_PRIMARY) ,OTU(FVR_800D_PRIMARY) ] ,XIO(FVR_800D_PRIMARY) [OTL(FVR_800D_PRIMARY) ,OTU(FVR_800C_PRIMARY) ] ] ];
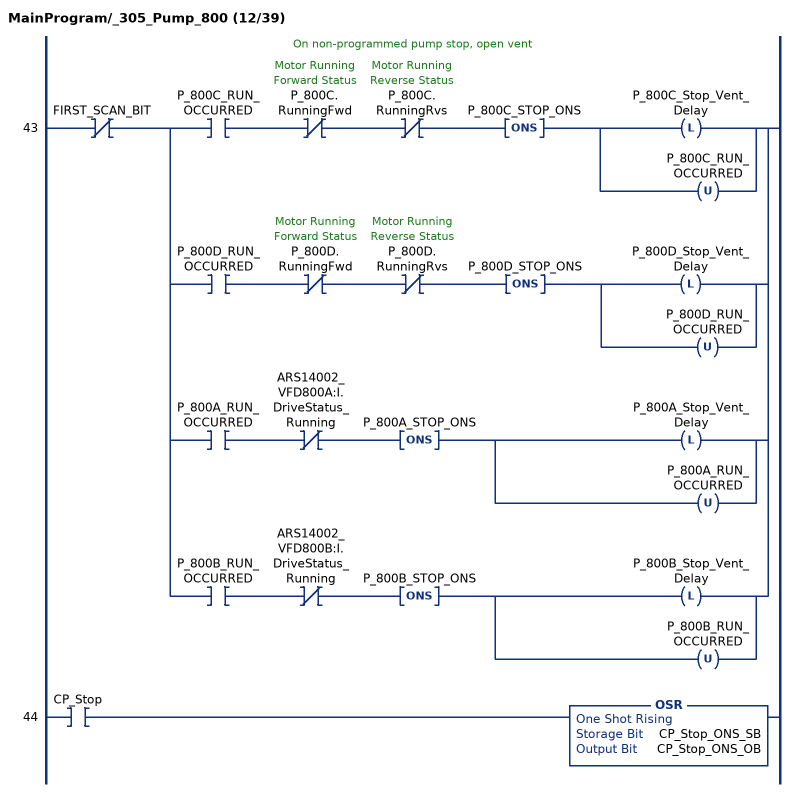
   // On non-programmed pump stop, open vent
   43: XIO(FIRST_SCAN_BIT)[XIC(P_800C_RUN_OCCURRED) XIO(P_800C.RunningFwd) XIO(P_800C.RunningRvs) ONS(P_800C_STOP_ONS) [OTL(P_800C_Stop_Vent_Delay) ,OTU(P_800C_RUN_OCCURRED) ] ,XIC(P_800D_RUN_OCCURRED) XIO(P_800D.RunningFwd) XIO(P_800D.RunningRvs) ONS(P_800D_STOP_ONS) [OTL(P_800D_Stop_Vent_Delay) ,OTU(P_800D_RUN_OCCURRED) ] ,XIC(P_800A_RUN_OCCURRED) XIO(ARS14002_VFD800A:I.DriveStatus_Running) ONS(P_800A_STOP_ONS) [OTL(P_800A_Stop_Vent_Delay) ,OTU(P_800A_RUN_OCCURRED) ] ,XIC(P_800B_RUN_OCCURRED) XIO(ARS14002_VFD800B:I.DriveStatus_Running) ONS(P_800B_STOP_ONS) [OTL(P_800B_Stop_Vent_Delay) ,OTU(P_800B_RUN_OCCURRED) ] ];
   44: XIC(CP_Stop)OSR(CP_Stop_ONS_SB,CP_Stop_ONS_OB);
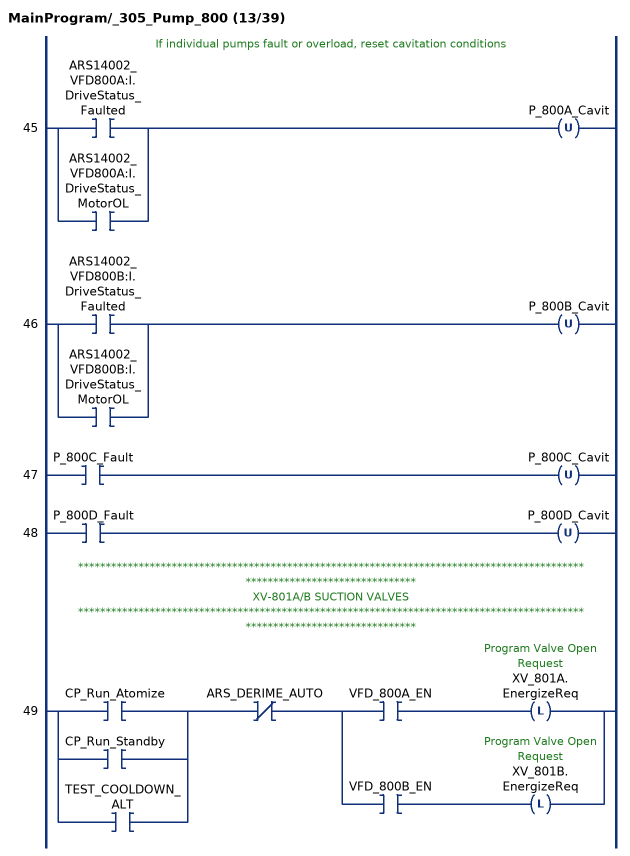
   // If individual pumps fault or overload, reset cavitation conditions
   45: [XIC(ARS14002_VFD800A:I.DriveStatus_Faulted) ,XIC(ARS14002_VFD800A:I.DriveStatus_MotorOL) ]OTU(P_800A_Cavit);
   46: [XIC(ARS14002_VFD800B:I.DriveStatus_Faulted) ,XIC(ARS14002_VFD800B:I.DriveStatus_MotorOL) ]OTU(P_800B_Cavit);
   47: XIC(P_800C_Fault)OTU(P_800C_Cavit);
   48: XIC(P_800D_Fault)OTU(P_800D_Cavit);
   // ***************************************************************************************************************************
   // XV-801A/B SUCTION VALVES
   // ***************************************************************************************************************************
   49: [XIC(CP_Run_Atomize) ,XIC(CP_Run_Standby) ,XIC(TEST_COOLDOWN_ALT) ]XIO(ARS_DERIME_AUTO)[XIC(VFD_800A_EN) OTL(XV_801A.EnergizeReq) ,XIC(VFD_800B_EN) OTL(XV_801B.EnergizeReq) ];
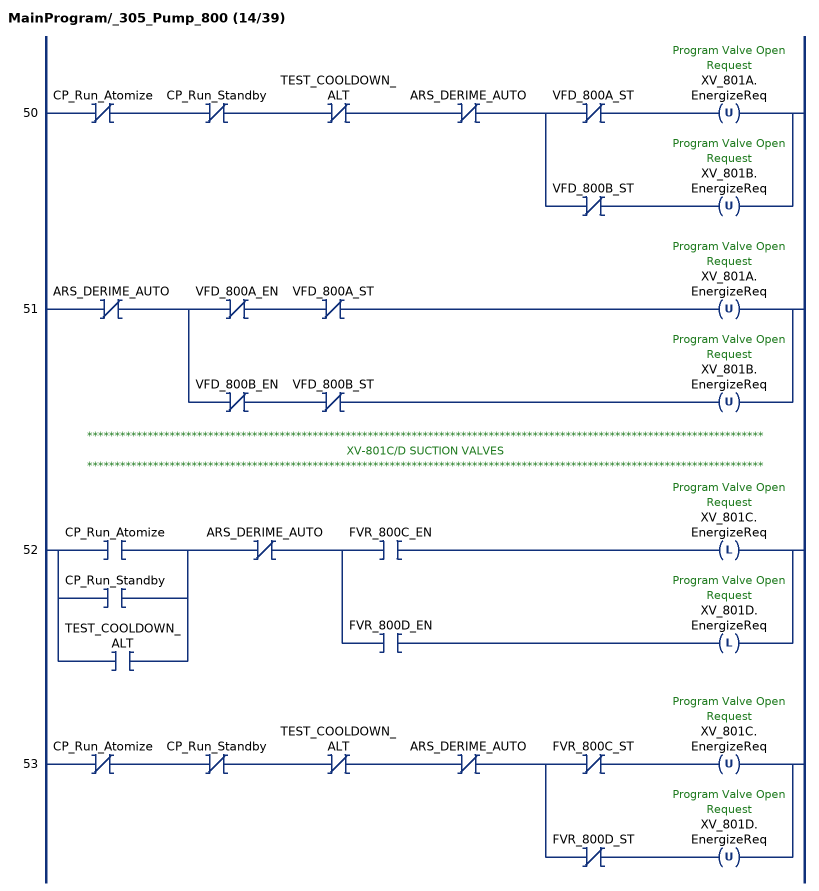
   50: XIO(CP_Run_Atomize)XIO(CP_Run_Standby)XIO(TEST_COOLDOWN_ALT)XIO(ARS_DERIME_AUTO)[XIO(VFD_800A_ST) OTU(XV_801A.EnergizeReq) ,XIO(VFD_800B_ST) OTU(XV_801B.EnergizeReq) ];
   51: XIO(ARS_DERIME_AUTO)[XIO(VFD_800A_EN) XIO(VFD_800A_ST) OTU(XV_801A.EnergizeReq) ,XIO(VFD_800B_EN) XIO(VFD_800B_ST) OTU(XV_801B.EnergizeReq) ];
   // ***************************************************************************************************************************
   // XV-801C/D SUCTION VALVES
   // ***************************************************************************************************************************
   52: [XIC(CP_Run_Atomize) ,XIC(CP_Run_Standby) ,XIC(TEST_COOLDOWN_ALT) ]XIO(ARS_DERIME_AUTO)[XIC(FVR_800C_EN) OTL(XV_801C.EnergizeReq) ,XIC(FVR_800D_EN) OTL(XV_801D.EnergizeReq) ];
   53: XIO(CP_Run_Atomize)XIO(CP_Run_Standby)XIO(TEST_COOLDOWN_ALT)XIO(ARS_DERIME_AUTO)[XIO(FVR_800C_ST) OTU(XV_801C.EnergizeReq) ,XIO(FVR_800D_ST) OTU(XV_801D.EnergizeReq) ];
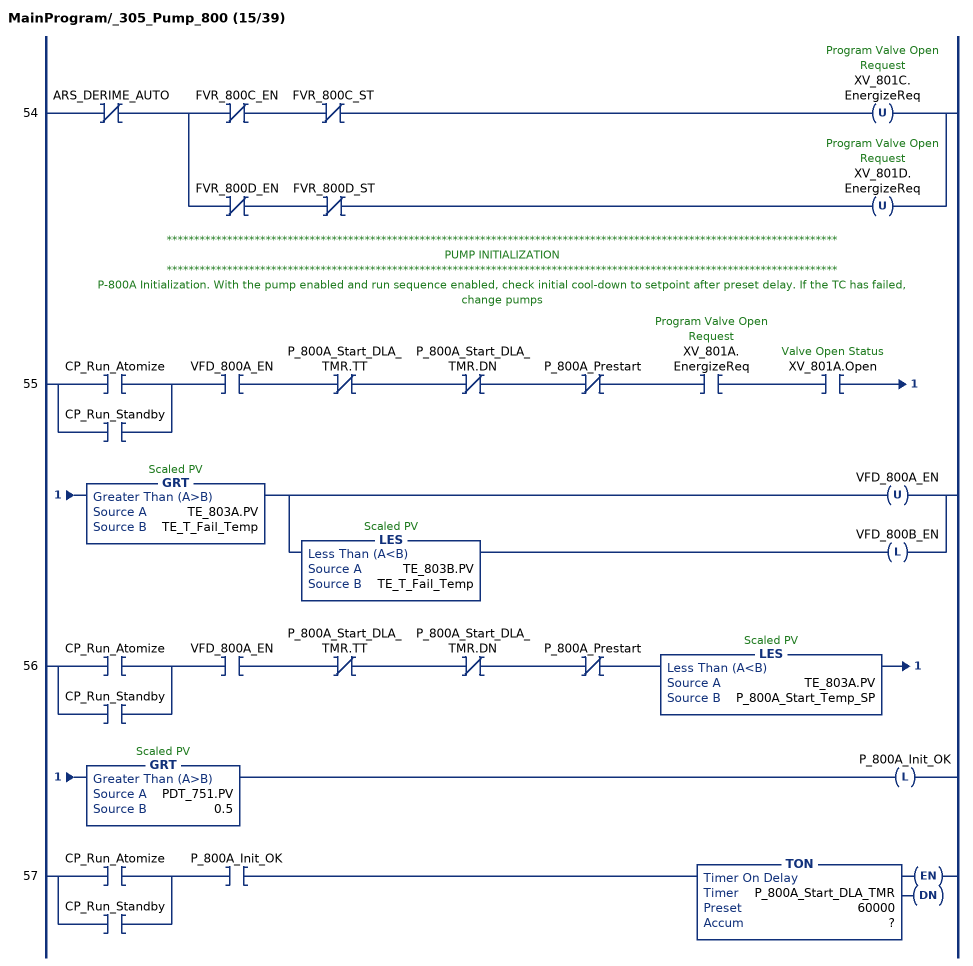
   54: XIO(ARS_DERIME_AUTO)[XIO(FVR_800C_EN) XIO(FVR_800C_ST) OTU(XV_801C.EnergizeReq) ,XIO(FVR_800D_EN) XIO(FVR_800D_ST) OTU(XV_801D.EnergizeReq) ];
   // **************************************************************************************************************************
   // PUMP INITIALIZATION
   // **************************************************************************************************************************
   // P-800A Initialization. With the pump enabled and run sequence enabled, check initial cool-down to setpoint after preset delay. If the TC has failed, change pumps
   55: [XIC(CP_Run_Atomize) ,XIC(CP_Run_Standby) ]XIC(VFD_800A_EN)XIO(P_800A_Start_DLA_TMR.TT)XIO(P_800A_Start_DLA_TMR.DN)XIO(P_800A_Prestart)XIC(XV_801A.EnergizeReq)XIC(XV_801A.Open)GRT(TE_803A.PV,TE_T_Fail_Temp)[OTU(VFD_800A_EN) ,LES(TE_803B.PV,TE_T_Fail_Temp) OTL(VFD_800B_EN) ];
   56: [XIC(CP_Run_Atomize) ,XIC(CP_Run_Standby) ]XIC(VFD_800A_EN)XIO(P_800A_Start_DLA_TMR.TT)XIO(P_800A_Start_DLA_TMR.DN)XIO(P_800A_Prestart)LES(TE_803A.PV,P_800A_Start_Temp_SP)GRT(PDT_751.PV,0.5)OTL(P_800A_Init_OK);
   57: [XIC(CP_Run_Atomize) ,XIC(CP_Run_Standby) ]XIC(P_800A_Init_OK)TON(P_800A_Start_DLA_TMR,?,?);
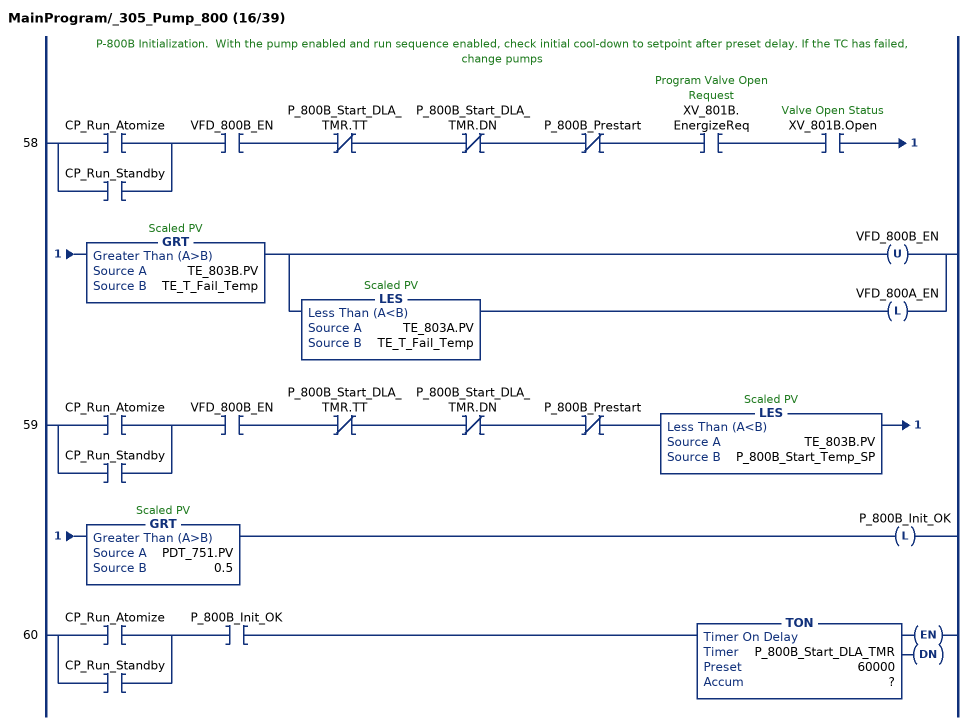
   // P-800B Initialization.  With the pump enabled and run sequence enabled, check initial cool-down to setpoint after preset delay. If the TC has failed, change pumps
   58: [XIC(CP_Run_Atomize) ,XIC(CP_Run_Standby) ]XIC(VFD_800B_EN)XIO(P_800B_Start_DLA_TMR.TT)XIO(P_800B_Start_DLA_TMR.DN)XIO(P_800B_Prestart)XIC(XV_801B.EnergizeReq)XIC(XV_801B.Open)GRT(TE_803B.PV,TE_T_Fail_Temp)[OTU(VFD_800B_EN) ,LES(TE_803A.PV,TE_T_Fail_Temp) OTL(VFD_800A_EN) ];
   59: [XIC(CP_Run_Atomize) ,XIC(CP_Run_Standby) ]XIC(VFD_800B_EN)XIO(P_800B_Start_DLA_TMR.TT)XIO(P_800B_Start_DLA_TMR.DN)XIO(P_800B_Prestart)LES(TE_803B.PV,P_800B_Start_Temp_SP)GRT(PDT_751.PV,0.5)OTL(P_800B_Init_OK);
   60: [XIC(CP_Run_Atomize) ,XIC(CP_Run_Standby) ]XIC(P_800B_Init_OK)TON(P_800B_Start_DLA_TMR,?,?);
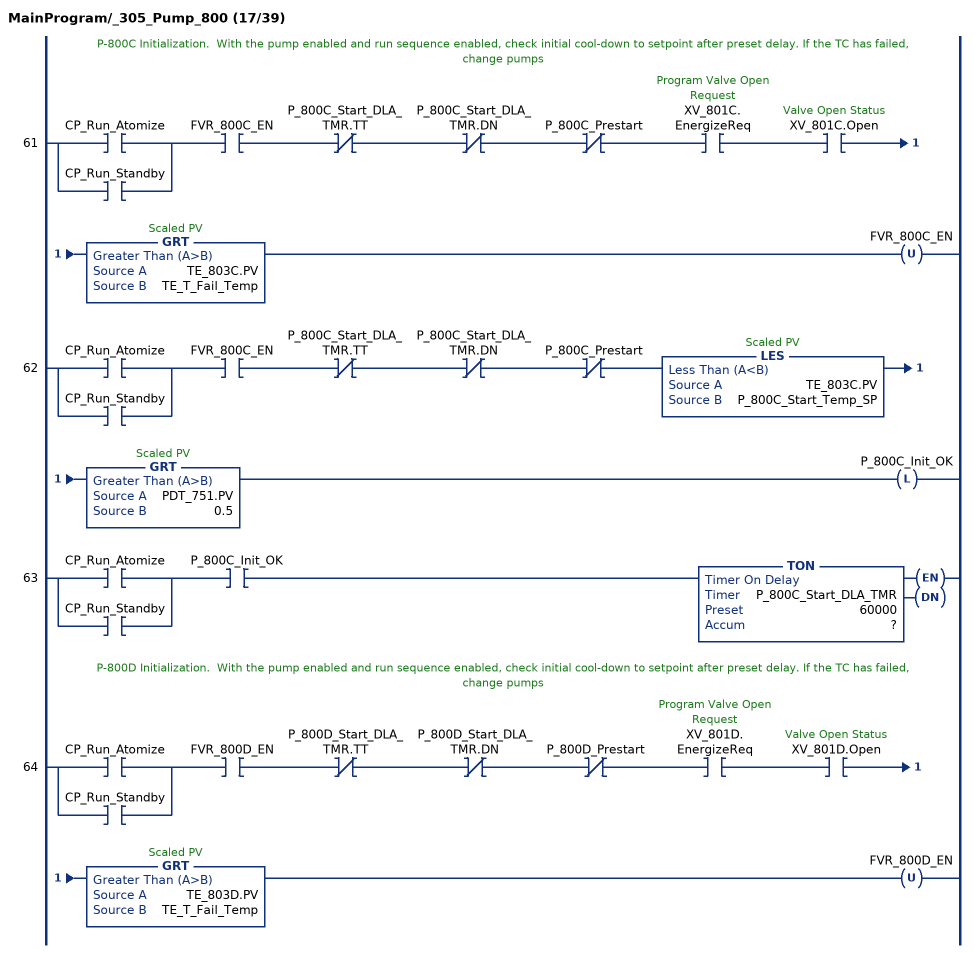
   // P-800C Initialization.  With the pump enabled and run sequence enabled, check initial cool-down to setpoint after preset delay. If the TC has failed, change pumps
   61: [XIC(CP_Run_Atomize) ,XIC(CP_Run_Standby) ]XIC(FVR_800C_EN)XIO(P_800C_Start_DLA_TMR.TT)XIO(P_800C_Start_DLA_TMR.DN)XIO(P_800C_Prestart)XIC(XV_801C.EnergizeReq)XIC(XV_801C.Open)GRT(TE_803C.PV,TE_T_Fail_Temp)OTU(FVR_800C_EN);
   62: [XIC(CP_Run_Atomize) ,XIC(CP_Run_Standby) ]XIC(FVR_800C_EN)XIO(P_800C_Start_DLA_TMR.TT)XIO(P_800C_Start_DLA_TMR.DN)XIO(P_800C_Prestart)LES(TE_803C.PV,P_800C_Start_Temp_SP)GRT(PDT_751.PV,0.5)OTL(P_800C_Init_OK);
   63: [XIC(CP_Run_Atomize) ,XIC(CP_Run_Standby) ]XIC(P_800C_Init_OK)TON(P_800C_Start_DLA_TMR,?,?);
   // P-800D Initialization.  With the pump enabled and run sequence enabled, check initial cool-down to setpoint after preset delay. If the TC has failed, change pumps
   64: [XIC(CP_Run_Atomize) ,XIC(CP_Run_Standby) ]XIC(FVR_800D_EN)XIO(P_800D_Start_DLA_TMR.TT)XIO(P_800D_Start_DLA_TMR.DN)XIO(P_800D_Prestart)XIC(XV_801D.EnergizeReq)XIC(XV_801D.Open)GRT(TE_803D.PV,TE_T_Fail_Temp)OTU(FVR_800D_EN);
